Staubli VAL3: handleNtype.pgx

program handleNtype()
  local bool l_bIsNumeric
  local num l_nTxtBoxVal
  local string l_sInputValue
begin
  // If attribute is Numeric,remove 0 from string
  if (pw:sTxtBoxType[nFocused]=="N")
    // Remove 0 if present
    if pw:sTxtBoxVal[nFocused]!="0"
      call _removeChar(pw:sTxtBoxVal[nFocused],"0",1,l_sInputValue)
    else
      l_sInputValue=pw:sTxtBoxVal[nFocused]
    endIf
    call _GetUserInput(l_sInputValue)
  endIf
  // If attribute is Numeric,check if value is in range
  if (pw:sTxtBoxType[nFocused]=="N")
    toNum(l_sInputValue,l_nTxtBoxVal,l_bIsNumeric)
    if l_bIsNumeric
      if (l_nTxtBoxVal<nTxtMinVal[nFocused]) or (l_nTxtBoxVal>nTxtMaxVal[nFocused])
        popUpMsg("Value must be in range of "+toString(".",nTxtMinVal[nFocused])+"->"+toString(".",nTxtMaxVal[nFocused]))
        call _writeTxtBoxVal(nFocused,nVIDEOINVERSED,"R")
      else
        // Remove 0 if present
        call _removeChar(l_sInputValue,"0",1,pw:sTxtBoxVal[nFocused])
        // force value to 0 if empty string
        if pw:sTxtBoxVal[nFocused]==""
          pw:sTxtBoxVal[nFocused]="0"
        endIf
      endIf
    else
      call _writeTxtBoxVal(nFocused,nVIDEOINVERSED,"R")
    endIf
    call _writeTxtBoxVal(nFocused,nVIDEOINVERSED,"R")
  endIf
end
